// :Description: Test-harness state (intentionally collides with Library.E_State to exercise ADR-0005's ambiguous-symbol error path).
TYPE E_State :
(
    Pending := 0,
    Pass := 1,
    Fail := 2
);
END_TYPE

(* stored: Version 1.1.0.1, ProductVersion 3.1.4026.0
   DUT E_State: Id {bbbbbbbb-bbbb-bbbb-bbbb-bbbbbbbbbbb3} *)
